PROGRAM MAIN
VAR
	bTestLightGreen:BOOL;
	bTestLightYellow:BOOL;
	bTestLightRed:BOOL;
END_VAR

END_PROGRAM

(* stored: Version 1.1.0.1, ProductVersion 3.1.4026.7
   POU MAIN: Id {26d3c236-5f98-4519-8342-39688ffe2109}, SpecialFunc None *)
